{attribute addProperty BoxType "AX2000-B110-0000"}
{attribute addProperty Id "Position_actual_valueAT %I*DINT3240Torque_actual_valueAT %I*INT1620Status_wordAT %I*UINT1620"}
{attribute addProperty CRC "892079825"}
{attribute addProperty SizeInBites "64"}
{attribute addProperty SizeInBytes "8"}
TYPE Inputs_352C0ED1 :
STRUCT
	{attribute addProperty Name "Position_actual_value"}
	Position_actual_value AT %I* : DINT;
	{attribute addProperty Name "Torque_actual_value"}
	Torque_actual_value AT %I* : INT;
	{attribute addProperty Name "Status_word"}
	Status_word AT %I* : UINT;
END_STRUCT
END_TYPE

(* stored: Version 1.2.0.0, ProductVersion 3.1.4024.9
   DUT Inputs_352C0ED1: Id {90ff4a5c-195b-432d-9d38-a5ddbec31abd} *)
